// TIA Portal V18 export
ORGANIZATION_BLOCK "Startup"   // OB100, LAD, Startup
TITLE = "Complete Restart"
{ S7_Optimized_Access := 'TRUE' }
// stored: SetENOAutomatically false
   VAR_INPUT
      LostRetentive : Bool;   // True if retentive data are lost
      LostRTC : Bool;   // True if date and time are lost
   END_VAR
   VAR_TEMP
      RetVal : Int;
      BusyStatus : Bool;
   END_VAR
   VAR_TEMP   // added for the SCL form of the ladder/FBD networks
      _w1 : Bool;
   END_VAR
BEGIN

REGION Network 1: Verify Settings
   // Check settings on startup
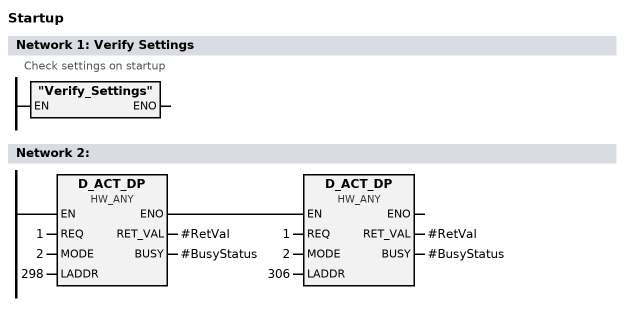
   RUNG wire#powerrail
      "Verify_Settings"()
   END_RUNG
   // the same network as SCL:
   "Verify_Settings"();
END_REGION

REGION Network 2
   RUNG wire#powerrail
      { S7_Templates := "[laddr_type := HW_ANY, mode_type := USInt]" } D_ACT_DP(REQ := 1, MODE := 2, LADDR := 298, RET_VAL => #RetVal, BUSY => #BusyStatus)
      { S7_Templates := "[laddr_type := HW_ANY, mode_type := USInt]" } D_ACT_DP(REQ := 1, MODE := 2, LADDR := 306, RET_VAL => #RetVal, BUSY => #BusyStatus)
   END_RUNG
   // the same network as SCL:
   #RetVal := D_ACT_DP(REQ := 1, MODE := 2, LADDR := 298, BUSY => #BusyStatus, ENO => #_w1);
   IF #_w1 THEN #RetVal := D_ACT_DP(REQ := 1, MODE := 2, LADDR := 306, BUSY => #BusyStatus); END_IF;
END_REGION
END_ORGANIZATION_BLOCK
